FUNCTION_BLOCK FB_Axis IMPLEMENTS I_Drivable
VAR
    bRunning : BOOL;
END_VAR

METHOD Start
bRunning := TRUE;
END_METHOD

END_FUNCTION_BLOCK

(* stored: Version 1.1.0.1, ProductVersion 3.1.4024.0
   POU FB_Axis: Id {7d2c9e41-5a86-4b0f-8c93-1e6d4a7b0c58}, SpecialFunc None
   Method Start: Id {a1f6c8e2-3b95-4d07-8a41-9c5e0f7a2b63} *)
